(* IEC 61131-3 sources: PLC-PDAM-Samarinda/Basic_Function, 3 files *)

(* ---- currentAnalogScaling.st ---- *)
FUNCTION_BLOCK currentAnalogScaling
VAR_INPUT
	iSensorValue : INT;
	sensorMaxValue : REAL;
	sensorMinValue : REAL;
    errorTresholdDown : INT;
    errorTresholdUp : INT;
END_VAR
VAR_OUTPUT
	error : WSTRING := errorCode;
	outValue :REAL := scalingValue;
END_VAR
VAR
	iRawValue : INT := iSensorValue;
	iMaxValue : INT;
	iMinValue : INT;
	sMaxValue : REAL :=sensorMaxValue;
	sMinValue : REAL :=sensorMinValue;
	scalingValue : REAL;
	errorSensor : BOOL;
	errorCode : WSTRING;
    errorTresDown : INT := errorTresholdDown;
    errorTresUp : INT := errorTresholdUp;
END_VAR

IF vRawValue < errorTresDown OR vRawValue > errorTresDown THEN
	errorSensor := TRUE;
	IF vRawValue < errorTresDown THEN
		errorCode := "Sensor disconnected, please check sensor";
		END_IF
	IF vRawValue > errorTresUp THEN
		errorCode := "Overcurrent, please check sensor";
		END_IF
ELSE
	scalingValue := (sMaxValue - sMinValue)/(vMaxValue - vMinValue) *(vRawValue - vMinValue);
END_IF

END_FUNCTION_BLOCK

(* ---- switchON.st ---- *)
FUNCTION_BLOCK switchON
VAR_INPUT
    power : BOOL;
END_VAR

VAR_OUTPUT
    status : BOOL :=load;
END_VAR

VAR
    state : BOOL := power;
    on : BOOL ;
    off : BOOL;
    load : BOOL;
END_VAR

IF state = TRUE THEN
    on := TRUE;
    off := FALSE;
    ELSE on := FALSE;
        off := TRUE;

//logic
load S= on;
load R=off

END_FUNCTION_BLOCK

(* ---- voltageAnalogScaling.st ---- *)
FUNCTION_BLOCK voltageAnalogScaling
VAR_INPUT
	vSensorValue : INT;
	sensorMaxValue : REAL;
	sensorMinValue : REAL;
    errorTresholdDown : INT;
    errorTresholdUp : INT;
END_VAR
VAR_OUTPUT
	error : WSTRING := errorCode;
	outValue :REAL := scalingValue;
END_VAR
VAR
	vRawValue : INT := iSensorValue;
	vMaxValue : INT;
	vMinValue : INT;
	sMaxValue : REAL :=sensorMaxValue;
	sMinValue : REAL :=sensorMinValue;
	scalingValue : REAL;
	errorSensor : BOOL;
	errorCode : WSTRING;
    errorTresDown : INT := errorTresholdDown;
    errorTresUp : INT := errorTresholdUp;
END_VAR

IF vRawValue < errorTresDown OR vRawValue > errorTresDown THEN
	errorSensor := TRUE;
	IF vRawValue < errorTresDown THEN
		errorCode := "Sensor disconnected, please check sensor";
		END_IF
	IF vRawValue > errorTresUp THEN
		errorCode := "Overcurrent, please check sensor";
		END_IF
ELSE
	scalingValue := (sMaxValue - sMinValue)/(vMaxValue - vMinValue) *(vRawValue - vMinValue);
END_IF

END_FUNCTION_BLOCK
